// TIA Portal V16 export
// export: Created 2026-06-18T08:51:49.8464013Z, ExportSetting WithDefaults, DisplayName Totally Integrated Automation Portal, DisplayVersion V16 Update 8, DisplayName TIA Portal Version Control Interface, DisplayVersion V16 Update 8, DisplayName TIA Portal Openness, DisplayVersion V16 Update 8, DisplayName SINAMICS Startdrive Advanced, DisplayVersion V16, DisplayName SINAMICS Startdrive G130, G150, S120, S150, SINAMICS MV, S210, DisplayVersion V16, DisplayName SINAMICS Startdrive G110M, G120, G120C, G120D, G120P, DisplayVersion V16, DisplayName STEP 7 Professional, DisplayVersion V16 Update 8, DisplayName STEP 7 Safety, DisplayVersion V16 Update 7, DisplayName WinCC Advanced, DisplayVersion V16 Update 8
Screen "Operator_Login"  800x480, Number=1
  ScreenLayer 
    IOField "IO_User" at 190,100 size 160x30  DataFormat=Decimal, FormatPattern=9999999, Mode=InOutput
    IOField "IO_Pass" at 190,150 size 160x30  DataFormat=Decimal, FormatPattern=9999999, Mode=InOutput
    SymbolicIOField "符号 I/O 域_1" at 177,87 size 170x32  CountVisibleItems=3, Mode=InOutput, OnValue=1, TextOff="0", TextOn="1"
    TextField "TXT_Title" at 200,20 size 400x40  Text="操作员登录"
    TextField "LMP_Online_lbl" at 550,121 size 42x22  Text="在线"
    TextField "TXT_Pass" at 100,150 size 80x30  Text="密码"
    TextField "TXT_User" at 100,100 size 80x30  Text="用户名"
    Button "BTN_Login" at 180,220 size 120x40  Mode=Text, TextOff="登录", TextOn="登录"
    Button "BTN_Logout" at 330,220 size 120x40  Mode=Text, TextOff="退出", TextOn="退出"
    Circle "LMP_Online" at 600,110 size 48x48
